FUNCTION_BLOCK fb_Test
VAR_INPUT
END_VAR
VAR_OUTPUT
	iCount : int;
END_VAR
VAR
END_VAR

iCount := iCount + 1;

END_FUNCTION_BLOCK

(* stored: Version 1.1.0.1, ProductVersion 3.1.4024.11
   POU fb_Test: Id {fd706bea-6946-439a-af9c-cac1aa70581d}, SpecialFunc None *)
